TYPE ST_RxXbox :
STRUCT
	counter : UDINT;
END_STRUCT
END_TYPE

(* stored: Version 1.1.0.1, ProductVersion 3.1.4022.7
   DUT ST_RxXbox: Id {42e8ce85-3cdf-47bf-a23a-d02b431ad435} *)
